FUNCTION_BLOCK ManualState IMPLEMENTS I_SD_ValveState
VAR_INPUT
END_VAR
VAR_OUTPUT
END_VAR
VAR
    _ptSdValve : POINTER TO SD_Valve;
    _transition : I_Transitive;
    delayTimer : Tc2_Standard.TP;
    command : BOOL;
END_VAR

delayTimer(IN:=command,PT:=T#5S);
IF command THEN
    command := FALSE;
END_IF

METHOD Close : BOOL
IF delayTimer.Q THEN
    Close := FALSE;
ELSE
    command := TRUE;
    Close := TRUE;
END_IF
END_METHOD

METHOD FB_init : BOOL
VAR_INPUT
	bInitRetains : BOOL; // if TRUE, the retain variables are initialized (warm start / cold start)
	bInCopyCode : BOOL;  // if TRUE, the instance afterwards gets moved into the copy code (online change)
    ptSdValve : POINTER TO SD_Valve;
END_VAR
_ptSdValve := ptSdValve;
END_METHOD

METHOD Open : BOOL
IF delayTimer.Q THEN
    Open := FALSE;
ELSE
    command := TRUE;
    Open := TRUE;
END_IF
END_METHOD

METHOD RUN
THIS^();
END_METHOD

METHOD SetTransition
VAR_INPUT
	transition	: I_Transitive;
END_VAR
_transition := transition;
END_METHOD

PROPERTY StateName : STRING
GET
StateName := 'Manual';
END_GET
END_PROPERTY

END_FUNCTION_BLOCK

(* stored: Version 1.1.0.1, ProductVersion 3.1.4024.12
   POU ManualState: Id {6c6f59f1-b7a2-4d13-804a-9a2a85fb3290}, SpecialFunc None
   Method Close: Id {73fffddb-f1f5-4b90-b0b4-e4392474250a}
   Method FB_init: Id {8b068cd2-7836-43e6-8f67-e64a62ae783c}
   Method Open: Id {6cf2b539-4c21-404d-b23c-88224b42aaed}
   Method RUN: Id {608798cb-2d01-412b-ac89-8219886bab1b}
   Method SetTransition: Id {6a0f7af4-5433-42fb-9172-2d714a0ad8ac}
   Property StateName: Id {2f1af59c-3b7c-4020-971c-df013ba1abe4}
   Get Get: Id {b28d3c98-25a2-4d8e-8592-024eef79e2f1} *)
